INTERFACE PUBLIC SuspendingCommands

METHOD PUBLIC Abort
END_METHOD

METHOD PUBLIC StateComplete
END_METHOD

METHOD PUBLIC Stop
END_METHOD

END_INTERFACE

(* stored: Version 1.1.0.1, ProductVersion 3.1.4026.12
   Itf SuspendingCommands: Id {293f49ed-8bfe-09e2-1376-339448adb778}
   Method Abort: Id {eeba19f4-7829-42de-8172-def3802d77b2}
   Method StateComplete: Id {718678b5-02aa-4eda-af48-80c3a021e43d}
   Method Stop: Id {9ebfdf27-b9c6-4d01-bc02-dec0c76bb3f5} *)
